{attribute 'linkalways'} 
{attribute 'no_explicit_call' := 'This FB is a CLASS and must be accessed using methods or properties'}
{attribute 'enable_dynamic_creation'}
FUNCTION_BLOCK ABSTRACT StructuredDatatypeBase EXTENDS UserDefinedDatatypeBase IMPLEMENTS I_StructuredDatatype
VAR
	membersHost : StructureMemberHost;
END_VAR

METHOD PUBLIC Accept
VAR_INPUT
	Visitor : I_DatatypeVisitor;
END_VAR
Visitor.VisitDatatype(THIS^);
membersHost.Accept(Visitor);
END_METHOD

METHOD PROTECTED AddMember
VAR_INPUT
	MemberName : T_MAXSTRING;
	Member : I_Datatype;
END_VAR
membersHost.AddMember(MemberName, Member);
END_METHOD

PROPERTY PUBLIC Members : I_StructureMembers
GET
Members := membersHost;
END_GET
END_PROPERTY

METHOD PROTECTED OnSerializeTypeWith
VAR_INPUT
	Serializer : I_Serializer;
END_VAR
SUPER^.OnSerializeTypeWith(Serializer);
membersHost.SerializeTypeWith(Serializer);
END_METHOD

METHOD PUBLIC SerializeWith
VAR_INPUT
	Serializer : I_Serializer;
END_VAR
Serializer.StartObject();
membersHost.SerializeWith(Serializer);
Serializer.EndObject();
END_METHOD

METHOD TryDeserializeFrom : BOOL
VAR_INPUT
	Deserializer : I_Deserializer;
	Feedback : I_DeserializerFeedback;
END_VAR
TryDeserializeFrom := membersHost.TryDeserializeFrom(Deserializer, Feedback);
END_METHOD

METHOD PUBLIC TryResolveAsStructuredDatatype : BOOL
VAR_INPUT
	Destination : REFERENCE TO I_StructuredDatatype;
END_VAR
Destination := THIS^;
TryResolveAsStructuredDatatype := TRUE;
END_METHOD

PROPERTY PUBLIC TypeName : T_MAXSTRING
GET
TypeName := 'STRUCT';
END_GET
END_PROPERTY

END_FUNCTION_BLOCK

(* stored: Version 1.1.0.1, ProductVersion 3.1.4024.13
   POU StructuredDatatypeBase: Id {bc150211-39c1-00b8-3052-dd0ac967ae97}, SpecialFunc None
   Folder Protected: Id {8a6cc4e9-0cf9-09ae-2600-c49f7b78b747}
   Method Accept: Id {2525fe4e-c2d7-023a-24ad-be353676dbec}
   Method AddMember: Id {995388ce-ce9f-07a0-3c1c-5a4b1c1db70b}
   Property Members: Id {e924424f-68fd-420c-bfcc-0c00d9c8ca5c}
   Get Get: Id {ea72665e-07db-45f6-a55b-a366cd94ac39}
   Method OnSerializeTypeWith: Id {9c6c9b2c-d674-0a1a-1c74-9c425d9519f1}
   Method SerializeWith: Id {e3b387e1-ec15-0ad5-11fd-34ceb26b6d8f}
   Method TryDeserializeFrom: Id {8f0213c3-fd2f-0a33-177e-22ac430367f1}
   Method TryResolveAsStructuredDatatype: Id {1c036e15-2be0-05af-3425-145ddbe4724f}
   Property TypeName: Id {bc10a3bf-cc5b-009c-23fd-26e2e5d92aaf}
   Get Get: Id {23cab9a1-ba8e-0b29-2f33-7ba99b4bdbfd} *)
